// SIMATIC S7-200 SMART project (STEP 7-Micro/WIN SMART), CPU SR30

ORGANIZATION_BLOCK 主程序:OB1
TITLE=程序注释
BEGIN
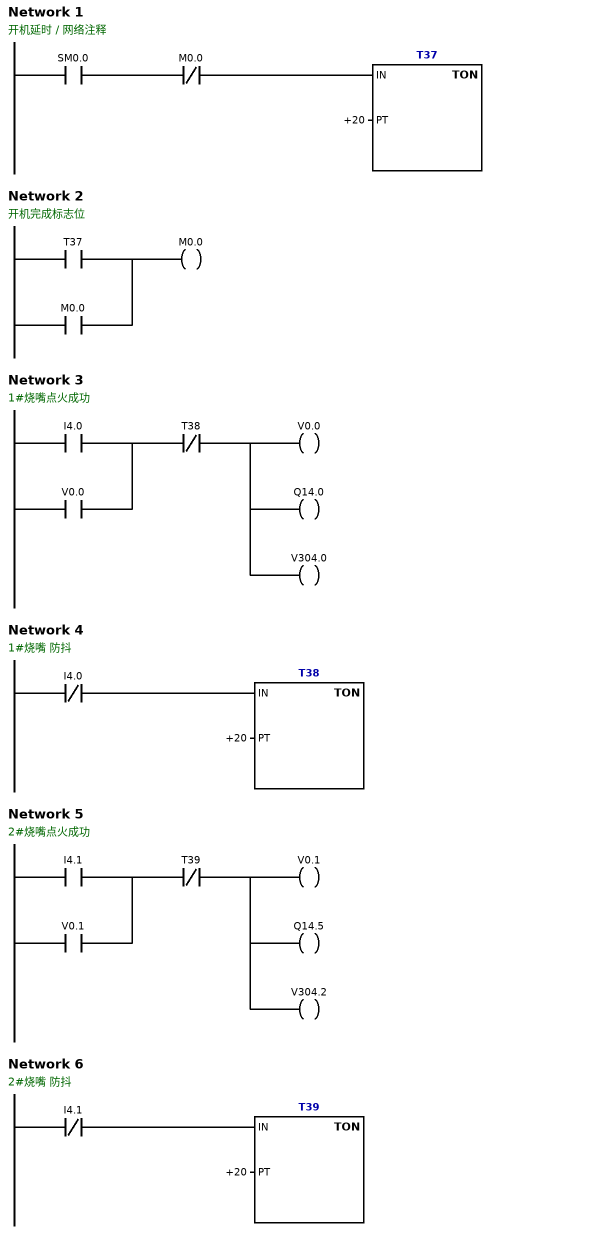
Network 1
// 开机延时
// 网络注释
LD     SM0.0
AN     M0.0
TON    T37, +20
Network 2
// 开机完成标志位
LD     T37
O      M0.0
=      M0.0
Network 3
// 1#烧嘴点火成功
LD     I4.0
O      V0.0
AN     T38
=      V0.0
=      Q14.0
=      V304.0
Network 4
// 1#烧嘴 防抖
LDN    I4.0
TON    T38, +20
Network 5
// 2#烧嘴点火成功
LD     I4.1
O      V0.1
AN     T39
=      V0.1
=      Q14.5
=      V304.2
Network 6
// 2#烧嘴 防抖
LDN    I4.1
TON    T39, +20
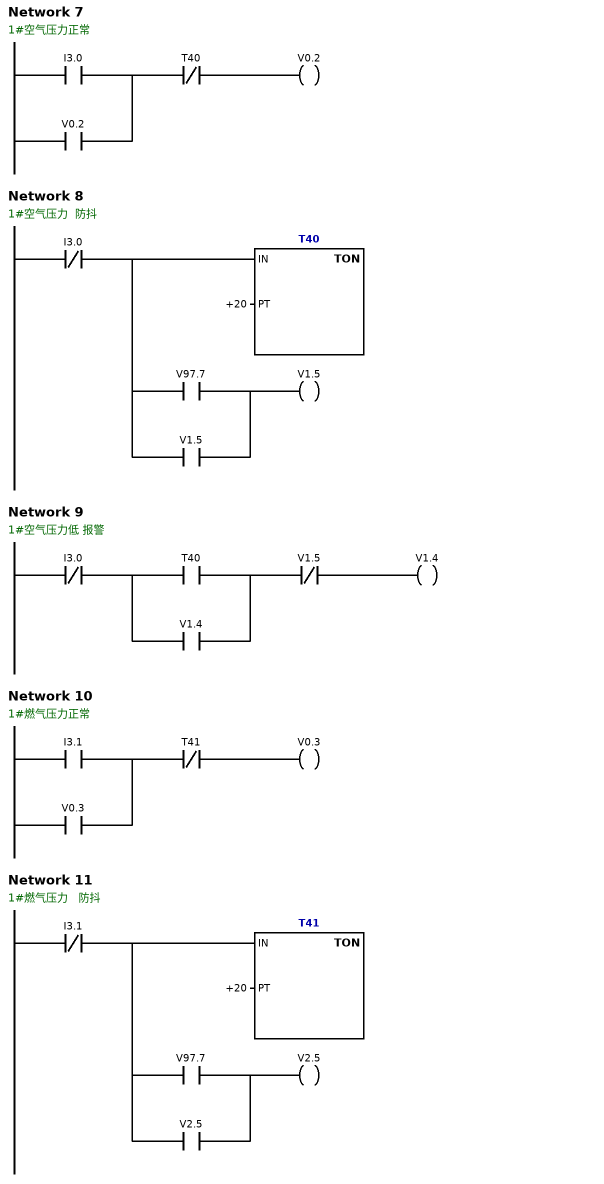
Network 7
// 1#空气压力正常
LD     I3.0
O      V0.2
AN     T40
=      V0.2
Network 8
// 1#空气压力  防抖
LDN    I3.0
TON    T40, +20
LD     V97.7
O      V1.5
ALD
=      V1.5
Network 9
// 1#空气压力低 报警
LDN    I3.0
LD     T40
O      V1.4
ALD
AN     V1.5
=      V1.4
Network 10
// 1#燃气压力正常
LD     I3.1
O      V0.3
AN     T41
=      V0.3
Network 11
// 1#燃气压力   防抖
LDN    I3.1
TON    T41, +20
LD     V97.7
O      V2.5
ALD
=      V2.5
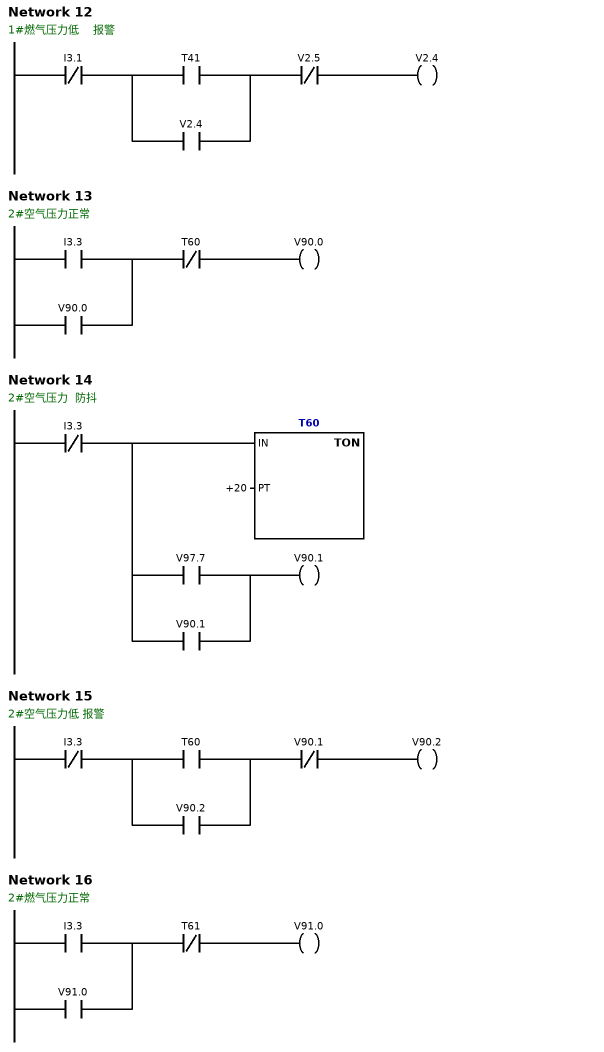
Network 12
// 1#燃气压力低    报警
LDN    I3.1
LD     T41
O      V2.4
ALD
AN     V2.5
=      V2.4
Network 13
// 2#空气压力正常
LD     I3.3
O      V90.0
AN     T60
=      V90.0
Network 14
// 2#空气压力  防抖
LDN    I3.3
TON    T60, +20
LD     V97.7
O      V90.1
ALD
=      V90.1
Network 15
// 2#空气压力低 报警
LDN    I3.3
LD     T60
O      V90.2
ALD
AN     V90.1
=      V90.2
Network 16
// 2#燃气压力正常
LD     I3.3
O      V91.0
AN     T61
=      V91.0
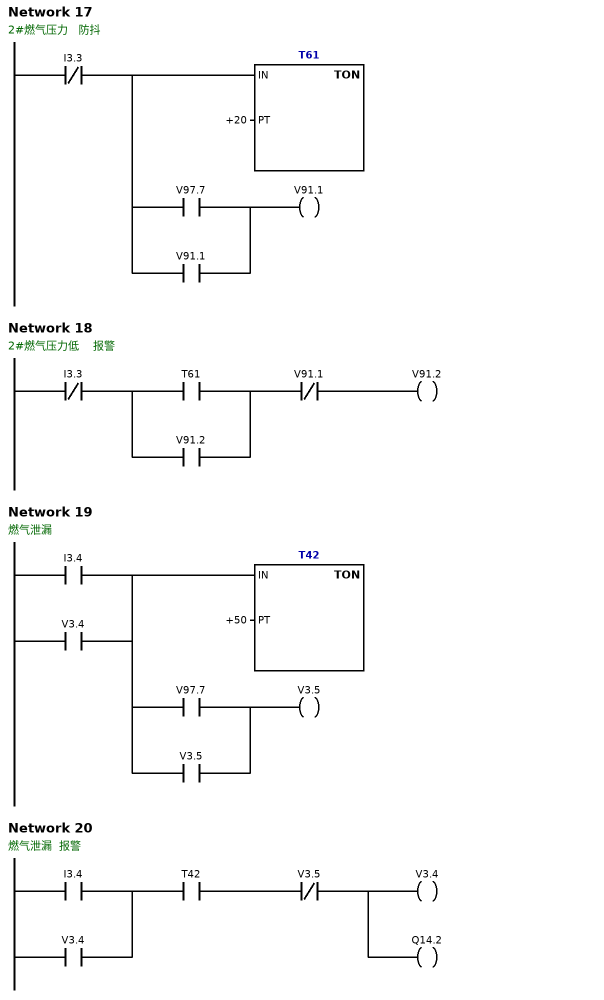
Network 17
// 2#燃气压力   防抖
LDN    I3.3
TON    T61, +20
LD     V97.7
O      V91.1
ALD
=      V91.1
Network 18
// 2#燃气压力低    报警
LDN    I3.3
LD     T61
O      V91.2
ALD
AN     V91.1
=      V91.2
Network 19
// 燃气泄漏
LD     I3.4
O      V3.4
TON    T42, +50
LD     V97.7
O      V3.5
ALD
=      V3.5
Network 20
// 燃气泄漏  报警
LD     I3.4
O      V3.4
A      T42
AN     V3.5
=      V3.4
=      Q14.2
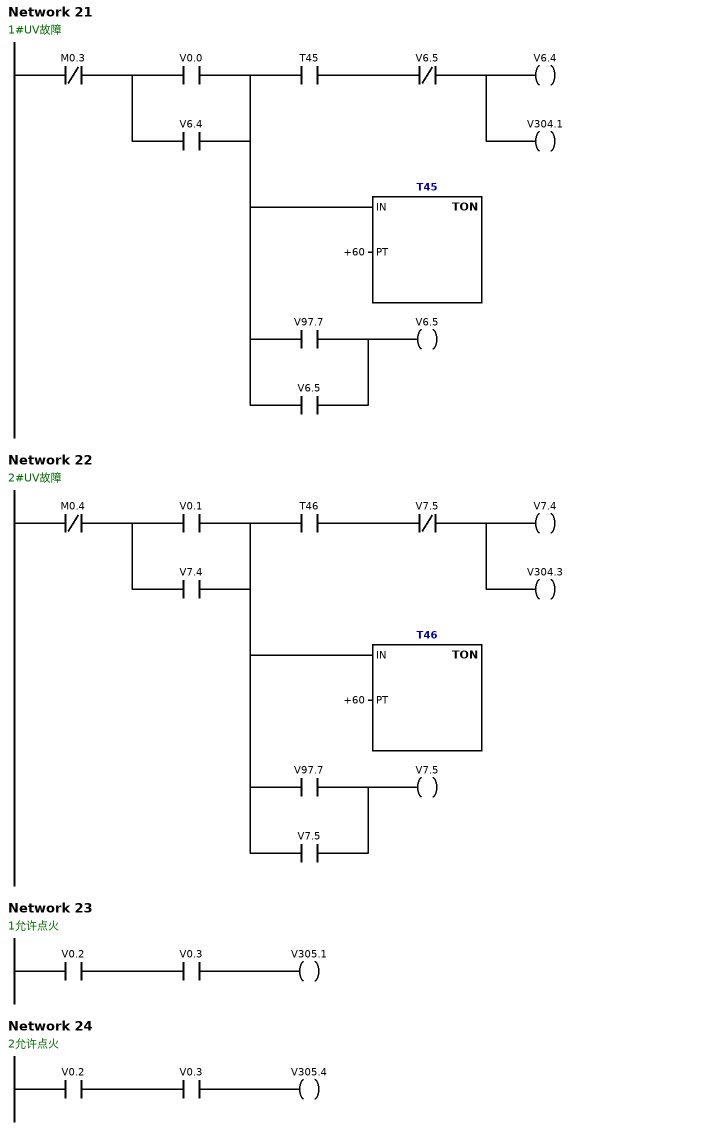
Network 21
// 1#UV故障
LDN    M0.3
LD     V0.0
O      V6.4
ALD
LPS
A      T45
AN     V6.5
=      V6.4
=      V304.1
LRD
TON    T45, +60
LPP
LD     V97.7
O      V6.5
ALD
=      V6.5
Network 22
// 2#UV故障
LDN    M0.4
LD     V0.1
O      V7.4
ALD
LPS
A      T46
AN     V7.5
=      V7.4
=      V304.3
LRD
TON    T46, +60
LPP
LD     V97.7
O      V7.5
ALD
=      V7.5
Network 23
// 1允许点火
// (network saved uncompiled; LAD cells follow)
// row 0: c0 -| |- V0.2  c1 -| |- V0.3  c2 -( ) V305.1
Network 24
// 2允许点火
// (network saved uncompiled; LAD cells follow)
// row 0: c0 -| |- V0.2  c1 -| |- V0.3  c2 -( ) V305.4
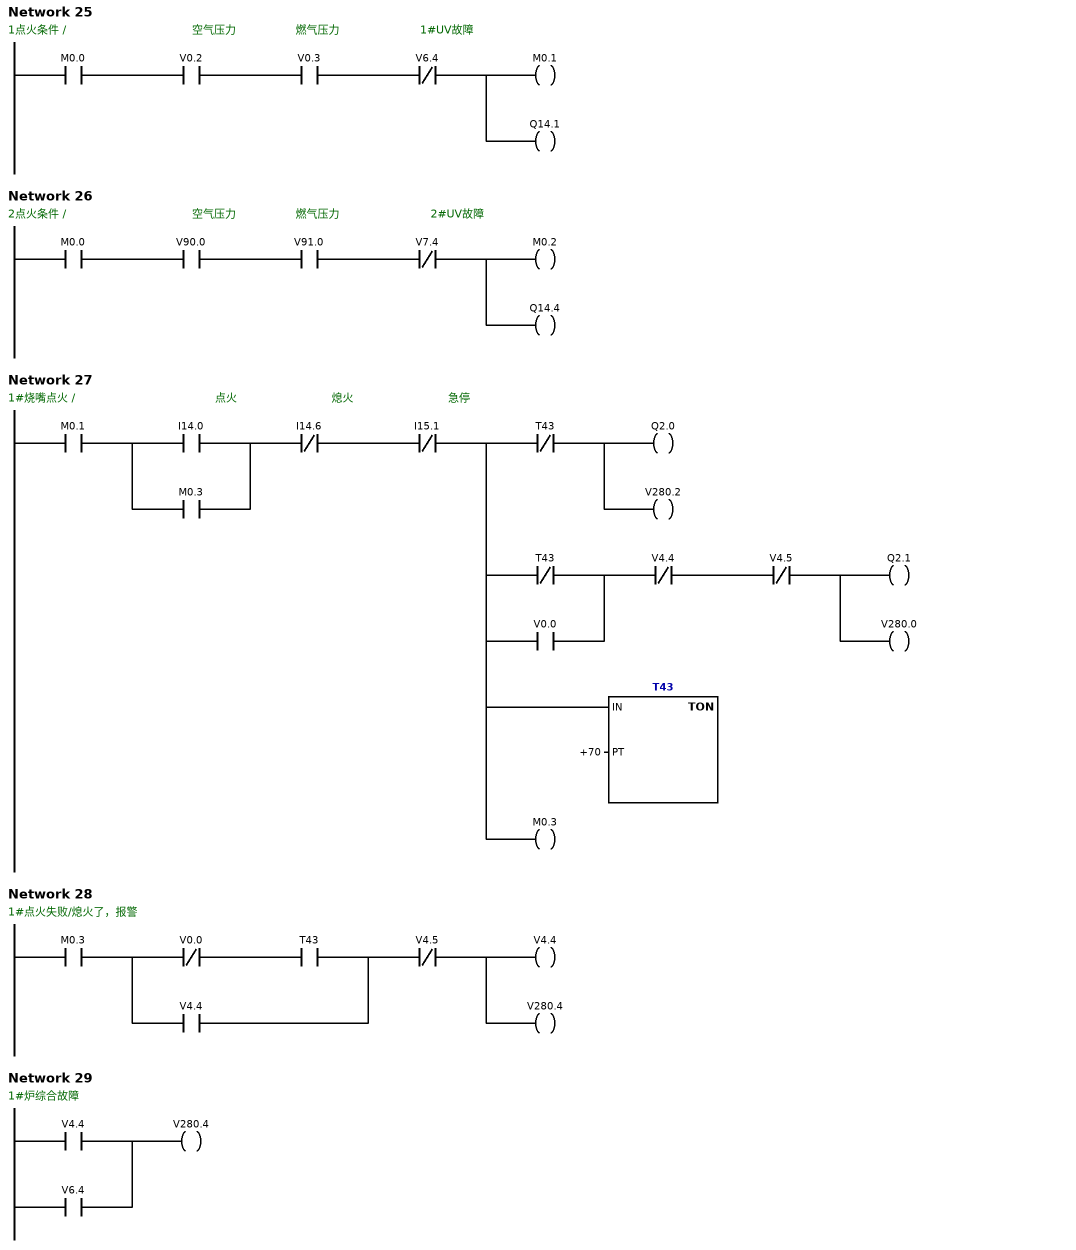
Network 25
// 1点火条件
//                                    空气压力                 燃气压力                       1#UV故障
LD     M0.0
A      V0.2
A      V0.3
AN     V6.4
=      M0.1
=      Q14.1
Network 26
// 2点火条件
//                                    空气压力                 燃气压力                          2#UV故障
LD     M0.0
A      V90.0
A      V91.0
AN     V7.4
=      M0.2
=      Q14.4
Network 27
// 1#烧嘴点火
//                                        点火                           熄火                           急停
LD     M0.1
LD     I14.0
O      M0.3
ALD
AN     I14.6
AN     I15.1
LPS
AN     T43
=      Q2.0
=      V280.2
LRD
LDN    T43
O      V0.0
AN     V4.4
AN     V4.5
ALD
=      Q2.1
=      V280.0
LPP
TON    T43, +70
=      M0.3
Network 28
// 1#点火失败/熄火了，报警
// (network saved uncompiled; LAD cells follow)
// row 0: c0 -| |- M0.3 v  c1 -|/|- V0.0  c2 -| |- T43 v  c3 -|/|- V4.5 v  c4 -( ) V4.4
// row 1: c0 ^  c1 -| |- V4.4  c2 -- ^  c3 ^  c4 -( ) V280.4
Network 29
// 1#炉综合故障
LD     V4.4
O      V6.4
=      V280.4
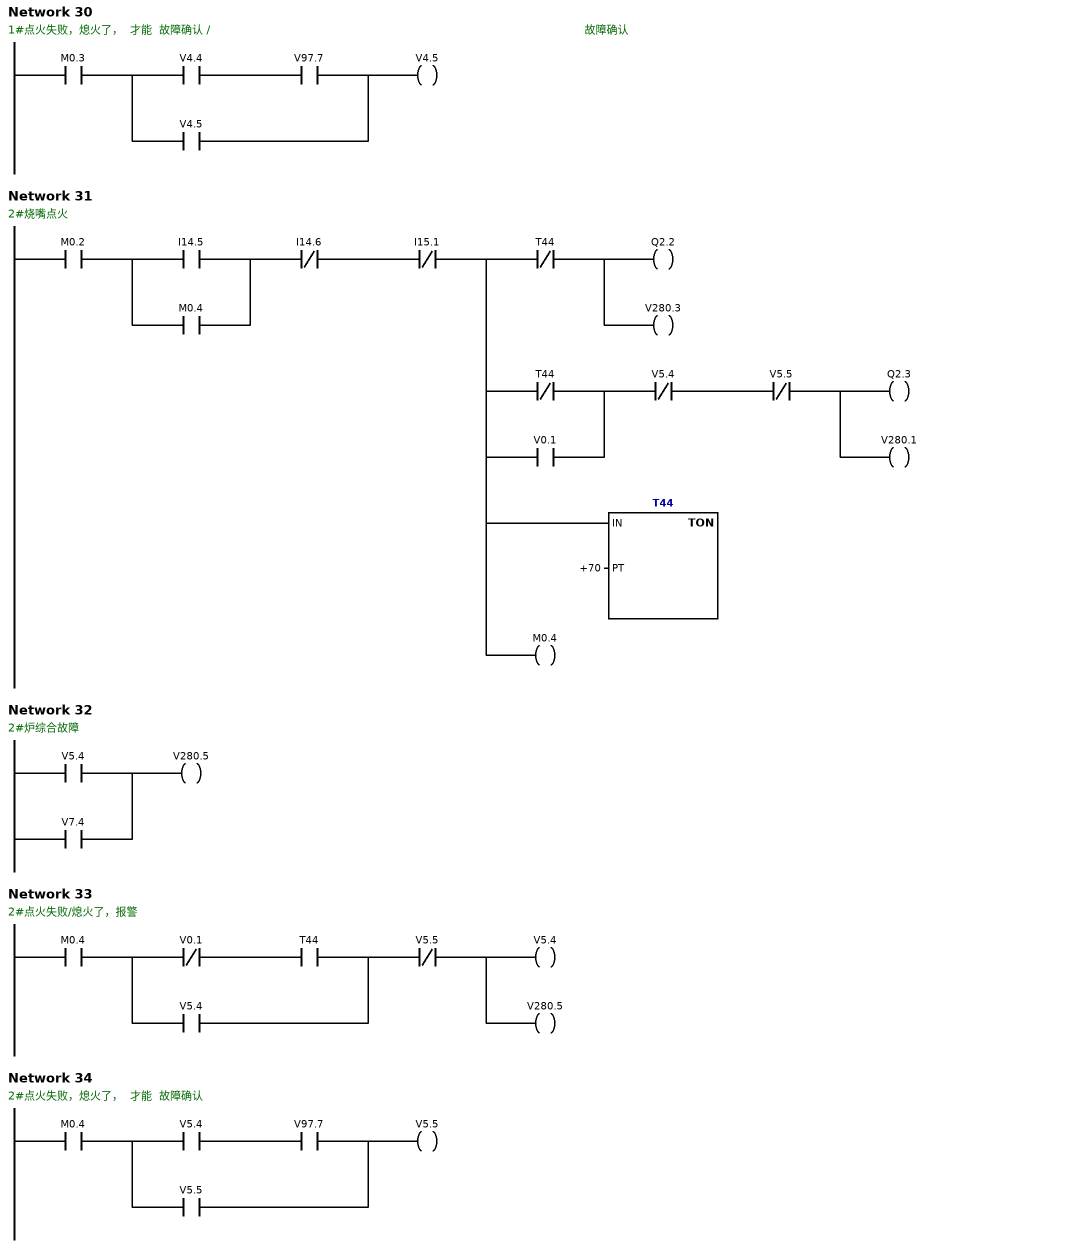
Network 30
// 1#点火失败，熄火了，  才能  故障确认
//                                                                                                           故障确认
LD     M0.3
LD     V4.4
A      V97.7
O      V4.5
ALD
=      V4.5
Network 31
// 2#烧嘴点火
// (network saved uncompiled; LAD cells follow)
// row 0: c0 -| |- M0.2 v  c1 -| |- I14.5 v  c2 -|/|- I14.6  c3 -|/|- I15.1 v  c4 -|/|- T44 v  c5 -( ) Q2.2
// row 1: c0 ^  c1 -| |- M0.4 ^  c3 ^v  c4 ^  c5 -( ) V280.3
// row 2: c3 ^v  c4 -|/|- T44 v  c5 -|/|- V5.4  c6 -|/|- V5.5 v  c7 -( ) Q2.3
// row 3: c3 ^v  c4 -| |- V0.1 ^  c6 ^  c7 -( ) V280.1
// row 4: c3 ^v  c4 --  c5 [TON T44 IN:=power@row4, PT:=+70]
// row 5: c3 ^v  c5 [box]
// row 6: c3 ^  c4 -( ) M0.4
Network 32
// 2#炉综合故障
LD     V5.4
O      V7.4
=      V280.5
Network 33
// 2#点火失败/熄火了，报警
// (network saved uncompiled; LAD cells follow)
// row 0: c0 -| |- M0.4 v  c1 -|/|- V0.1  c2 -| |- T44 v  c3 -|/|- V5.5 v  c4 -( ) V5.4
// row 1: c0 ^  c1 -| |- V5.4  c2 -- ^  c3 ^  c4 -( ) V280.5
Network 34
// 2#点火失败，熄火了，  才能  故障确认
LD     M0.4
LD     V5.4
A      V97.7
O      V5.5
ALD
=      V5.5
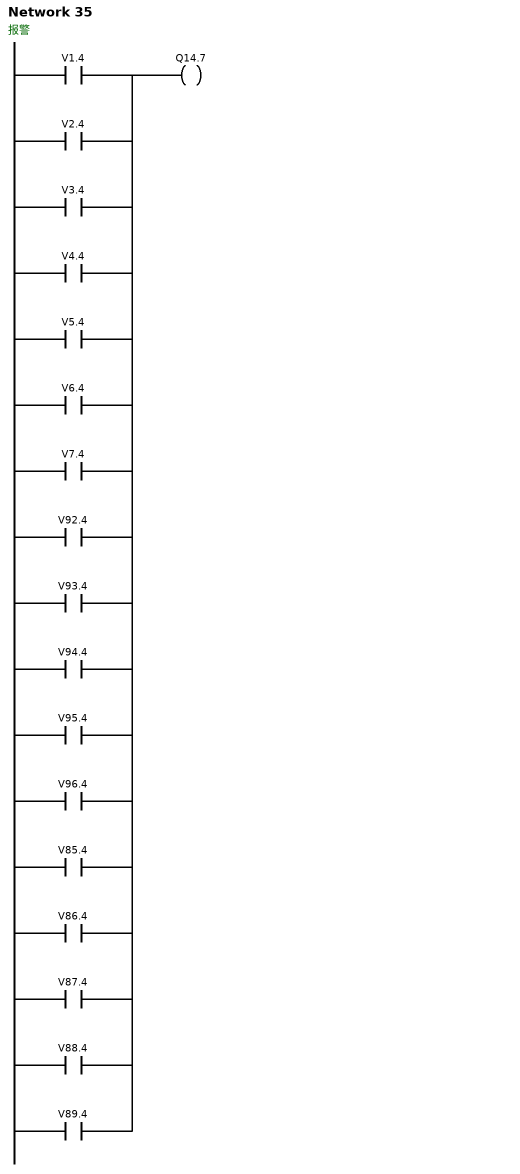
Network 35
// 报警
LD     V1.4
O      V2.4
O      V3.4
O      V4.4
O      V5.4
O      V6.4
O      V7.4
O      V92.4
O      V93.4
O      V94.4
O      V95.4
O      V96.4
O      V85.4
O      V86.4
O      V87.4
O      V88.4
O      V89.4
=      Q14.7
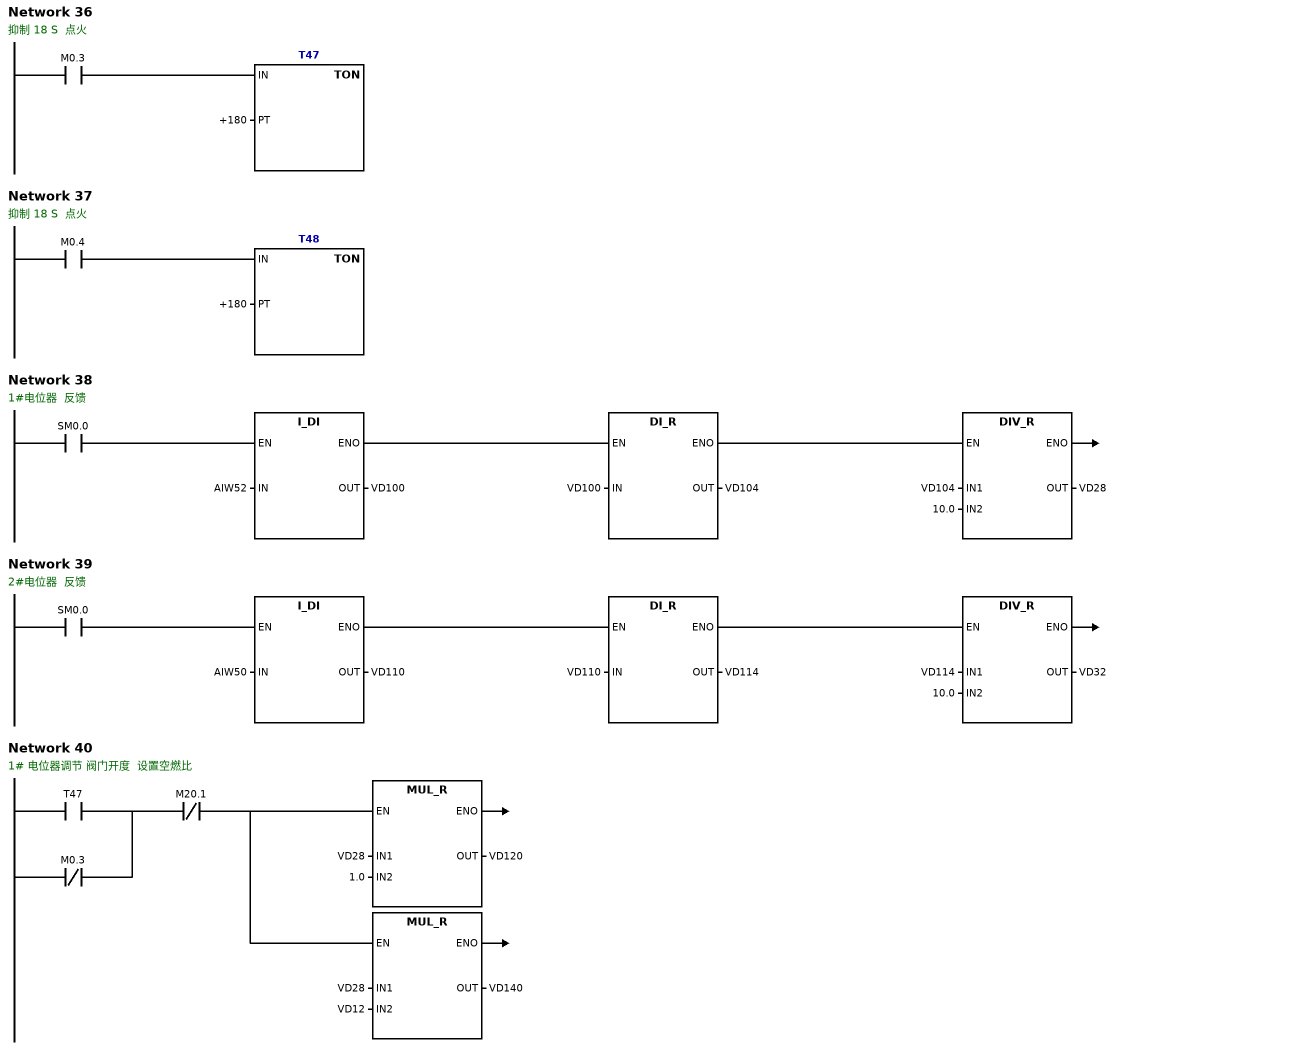
Network 36
// 抑制 18 S  点火
LD     M0.3
TON    T47, +180
Network 37
// 抑制 18 S  点火
LD     M0.4
TON    T48, +180
Network 38
// 1#电位器  反馈
LD     SM0.0
ITD    AIW52, VD100
AENO
DTR    VD100, VD104
AENO
MOVR   VD104, VD28
/R     10.0, VD28
Network 39
// 2#电位器  反馈
LD     SM0.0
ITD    AIW50, VD110
AENO
DTR    VD110, VD114
AENO
MOVR   VD114, VD32
/R     10.0, VD32
Network 40
// 1# 电位器调节 阀门开度  设置空燃比
LD     T47
ON     M0.3
AN     M20.1
MOVR   VD28, VD120
*R     1.0, VD120
MOVR   VD28, VD140
*R     VD12, VD140
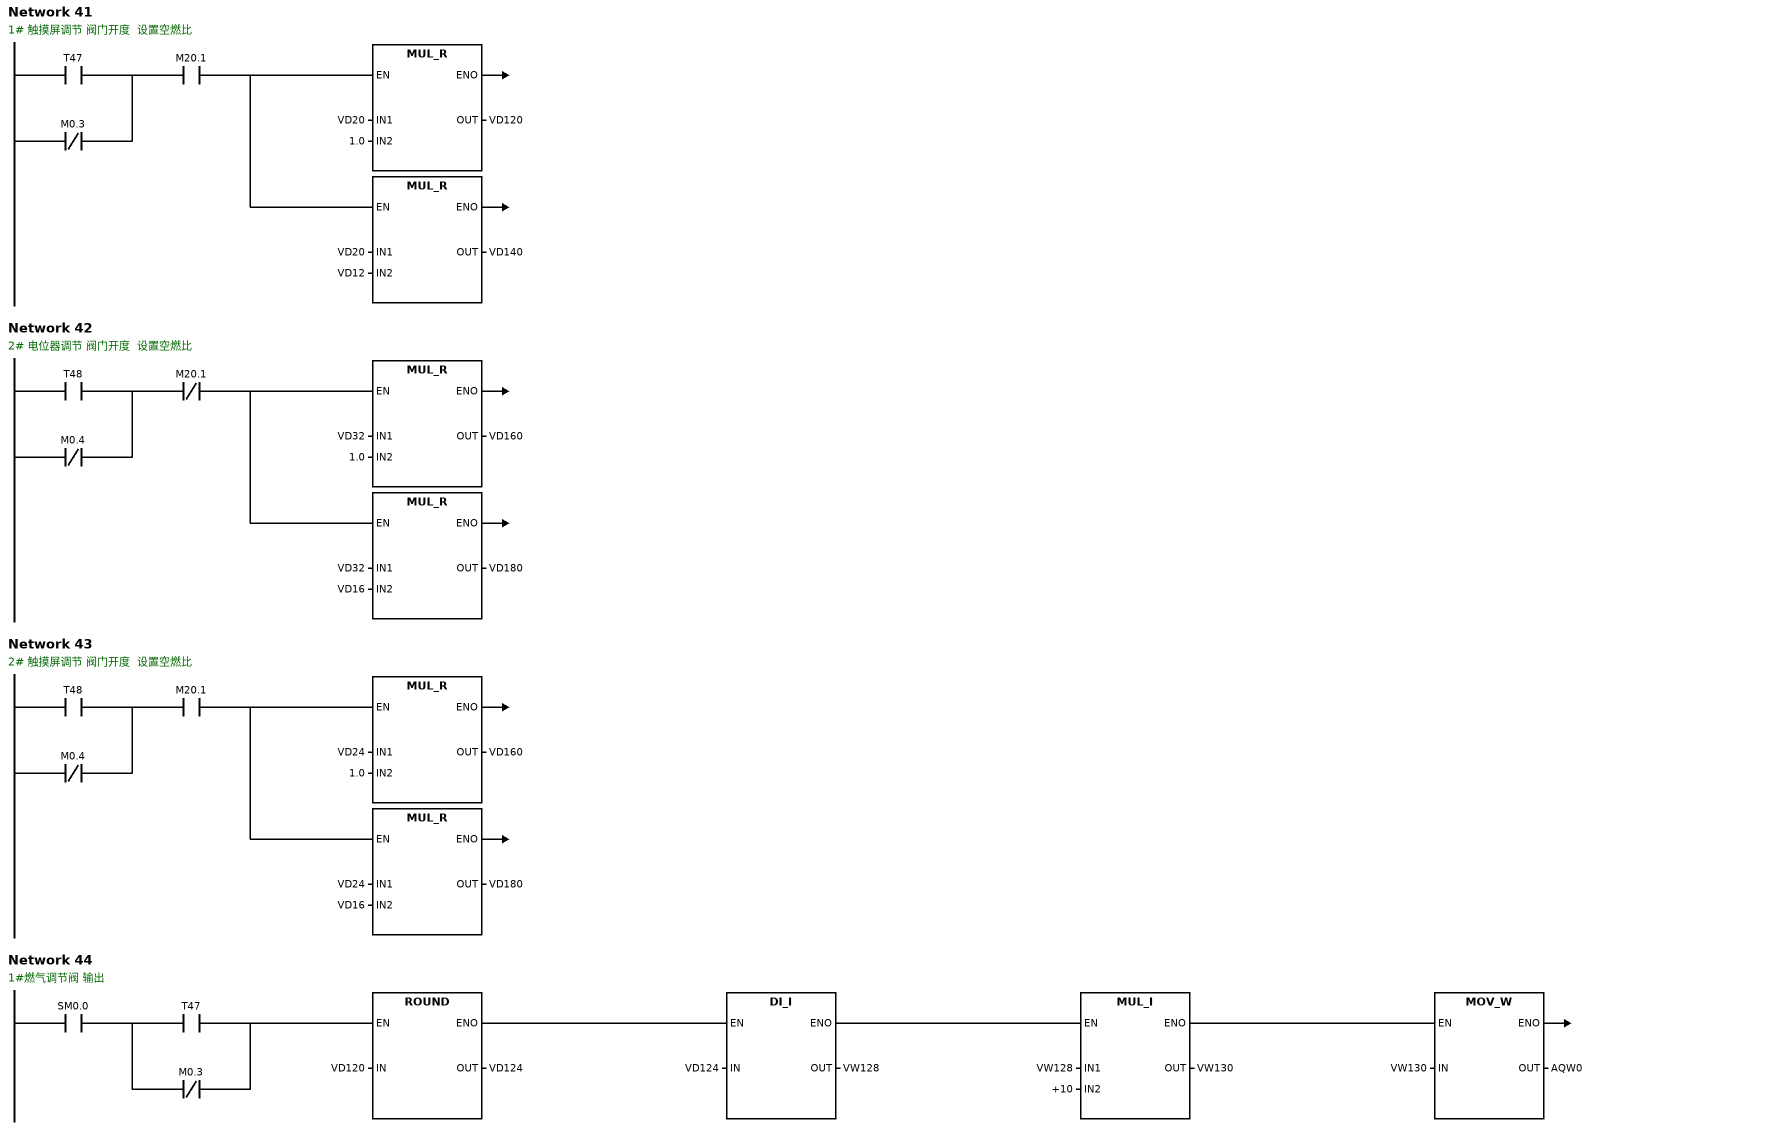
Network 41
// 1# 触摸屏调节 阀门开度  设置空燃比
LD     T47
ON     M0.3
A      M20.1
MOVR   VD20, VD120
*R     1.0, VD120
MOVR   VD20, VD140
*R     VD12, VD140
Network 42
// 2# 电位器调节 阀门开度  设置空燃比
LD     T48
ON     M0.4
AN     M20.1
MOVR   VD32, VD160
*R     1.0, VD160
MOVR   VD32, VD180
*R     VD16, VD180
Network 43
// 2# 触摸屏调节 阀门开度  设置空燃比
LD     T48
ON     M0.4
A      M20.1
MOVR   VD24, VD160
*R     1.0, VD160
MOVR   VD24, VD180
*R     VD16, VD180
Network 44
// 1#燃气调节阀 输出
LD     SM0.0
LD     T47
ON     M0.3
ALD
ROUND  VD120, VD124
AENO
DTI    VD124, VW128
AENO
MOVW   VW128, VW130
AENO
*I     +10, VW130
AENO
MOVW   VW130, AQW0
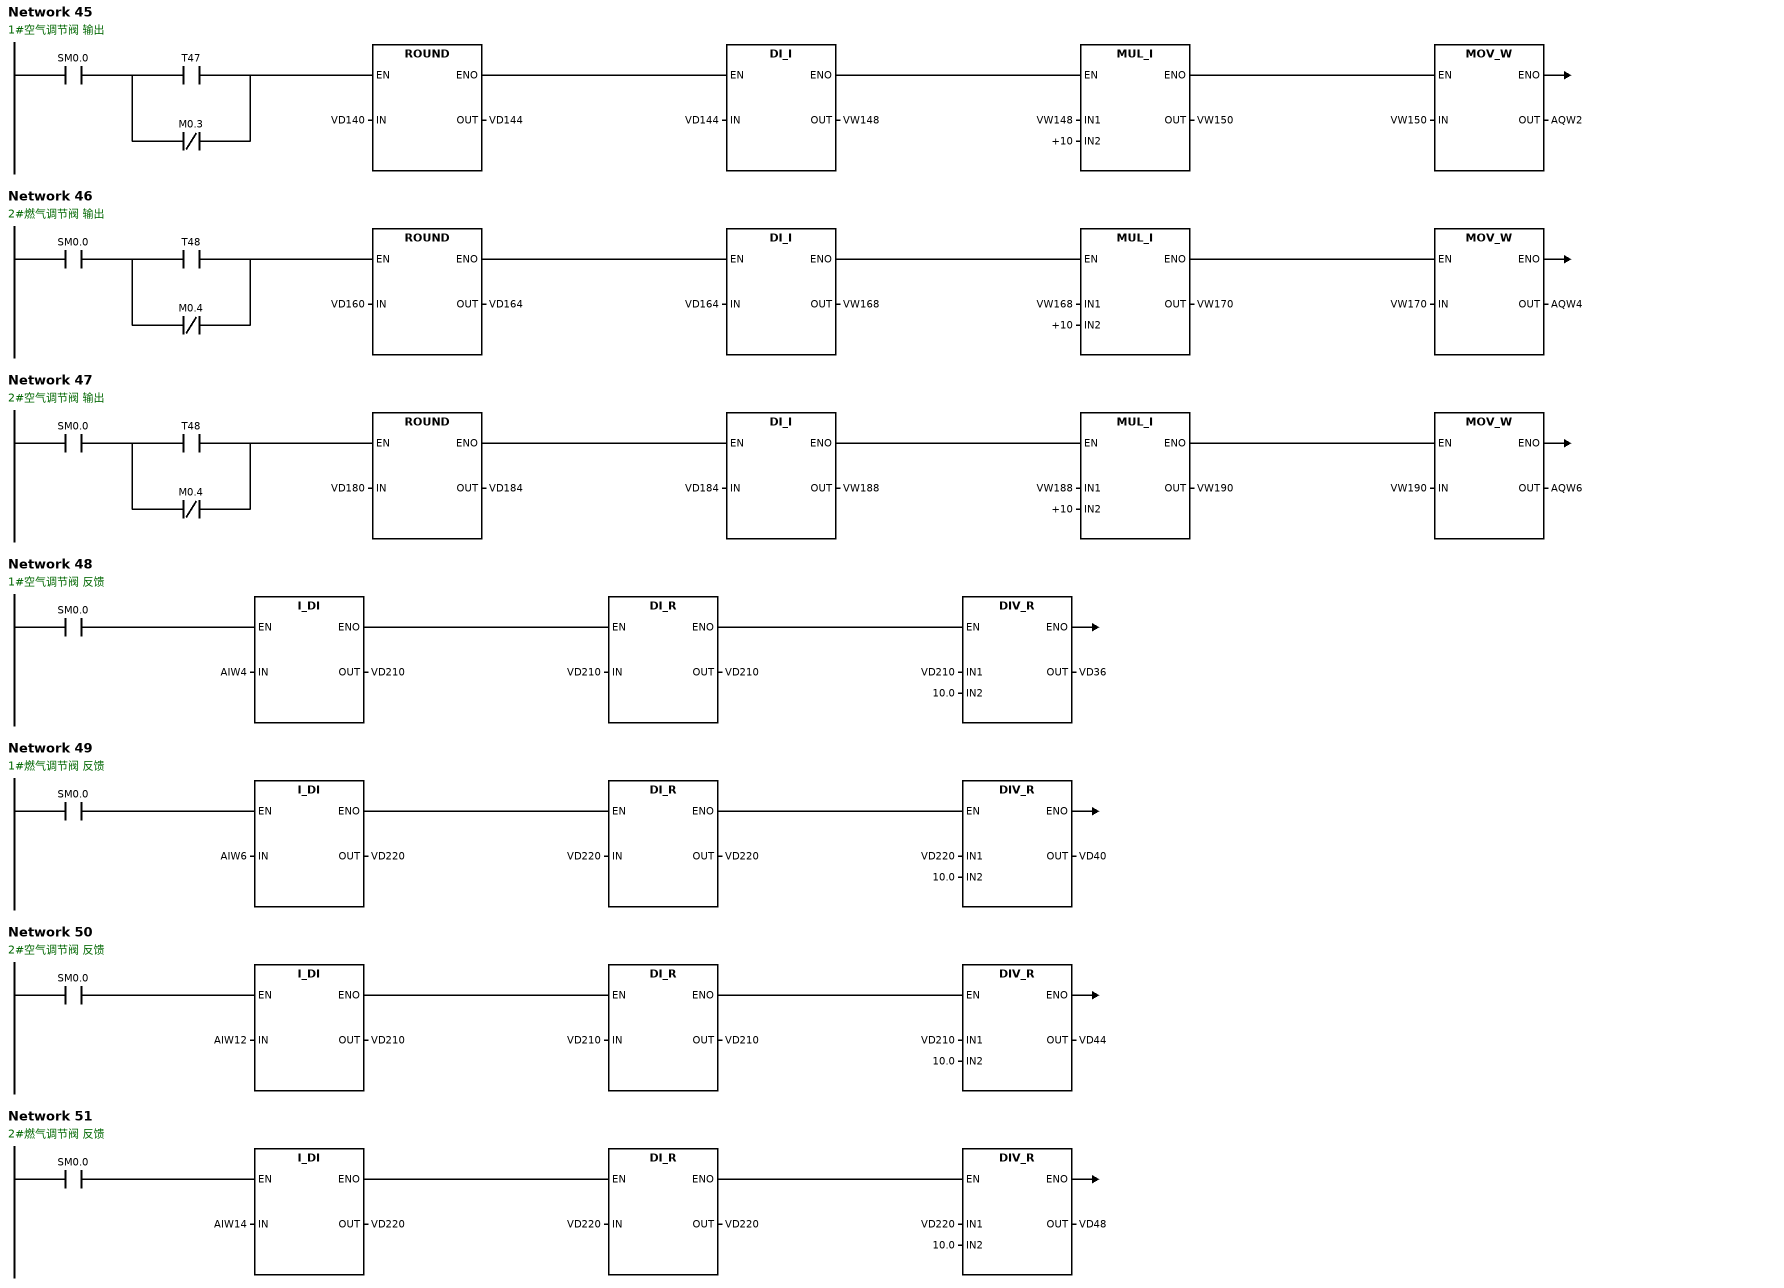
Network 45
// 1#空气调节阀 输出
LD     SM0.0
LD     T47
ON     M0.3
ALD
ROUND  VD140, VD144
AENO
DTI    VD144, VW148
AENO
MOVW   VW148, VW150
AENO
*I     +10, VW150
AENO
MOVW   VW150, AQW2
Network 46
// 2#燃气调节阀 输出
LD     SM0.0
LD     T48
ON     M0.4
ALD
ROUND  VD160, VD164
AENO
DTI    VD164, VW168
AENO
MOVW   VW168, VW170
AENO
*I     +10, VW170
AENO
MOVW   VW170, AQW4
Network 47
// 2#空气调节阀 输出
LD     SM0.0
LD     T48
ON     M0.4
ALD
ROUND  VD180, VD184
AENO
DTI    VD184, VW188
AENO
MOVW   VW188, VW190
AENO
*I     +10, VW190
AENO
MOVW   VW190, AQW6
Network 48
// 1#空气调节阀 反馈
LD     SM0.0
ITD    AIW4, VD210
AENO
DTR    VD210, VD210
AENO
MOVR   VD210, VD36
/R     10.0, VD36
Network 49
// 1#燃气调节阀 反馈
LD     SM0.0
ITD    AIW6, VD220
AENO
DTR    VD220, VD220
AENO
MOVR   VD220, VD40
/R     10.0, VD40
Network 50
// 2#空气调节阀 反馈
LD     SM0.0
ITD    AIW12, VD210
AENO
DTR    VD210, VD210
AENO
MOVR   VD210, VD44
/R     10.0, VD44
Network 51
// 2#燃气调节阀 反馈
LD     SM0.0
ITD    AIW14, VD220
AENO
DTR    VD220, VD220
AENO
MOVR   VD220, VD48
/R     10.0, VD48
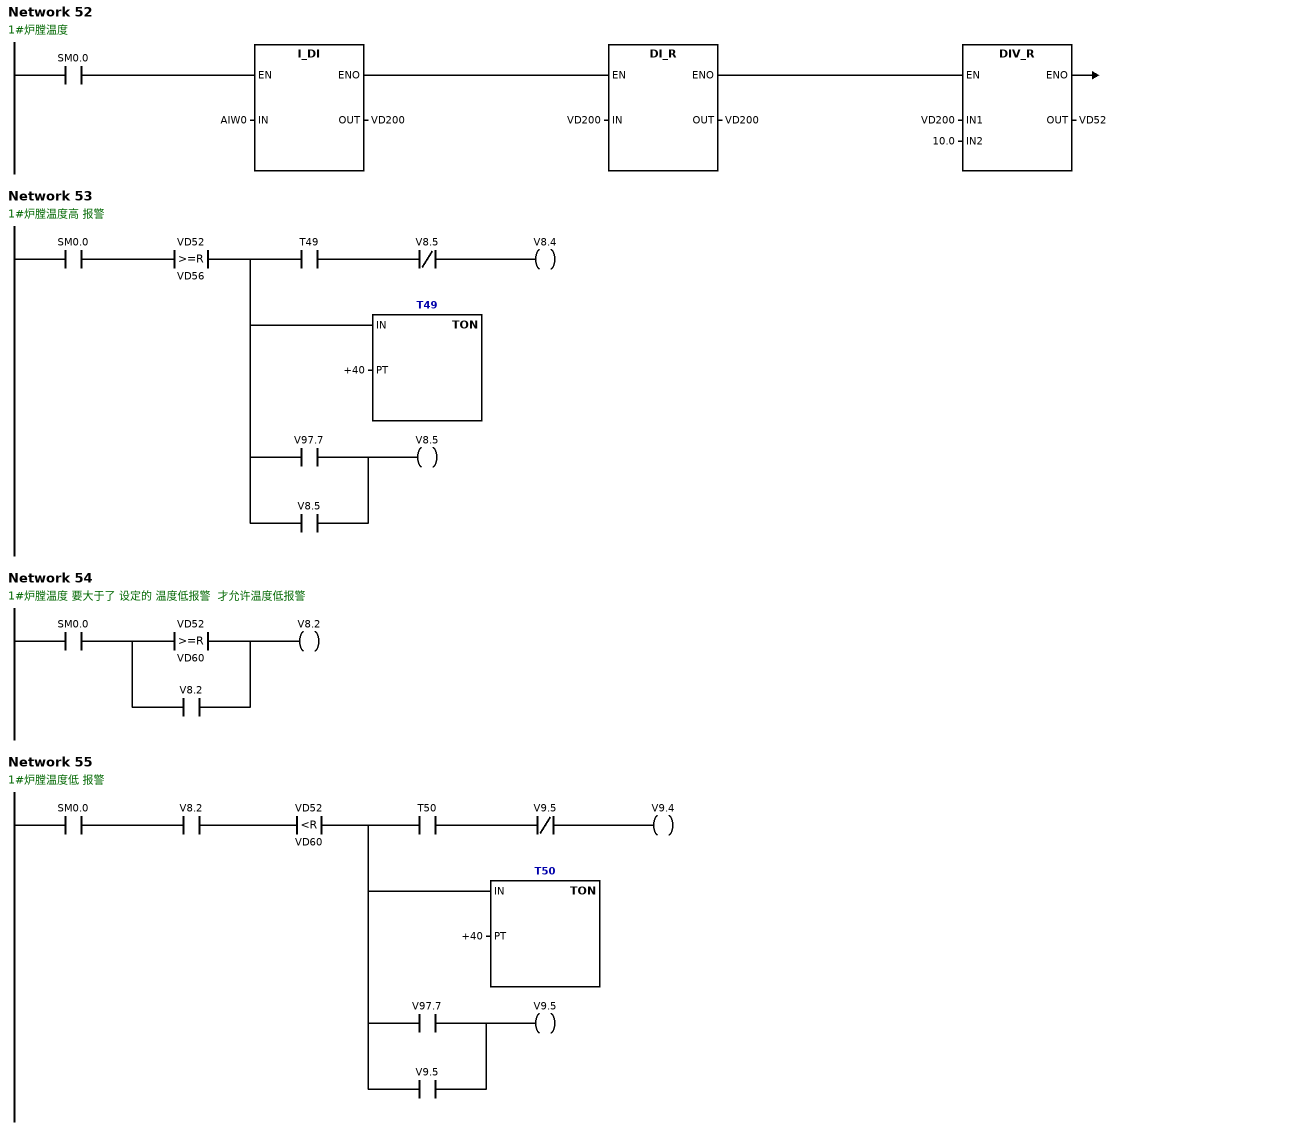
Network 52
// 1#炉膛温度
LD     SM0.0
ITD    AIW0, VD200
AENO
DTR    VD200, VD200
AENO
MOVR   VD200, VD52
/R     10.0, VD52
Network 53
// 1#炉膛温度高 报警
LD     SM0.0
AR>=   VD52, VD56
LPS
A      T49
AN     V8.5
=      V8.4
LRD
TON    T49, +40
LPP
LD     V97.7
O      V8.5
ALD
=      V8.5
Network 54
// 1#炉膛温度 要大于了 设定的 温度低报警  才允许温度低报警
LD     SM0.0
LDR>=  VD52, VD60
O      V8.2
ALD
=      V8.2
Network 55
// 1#炉膛温度低 报警
LD     SM0.0
A      V8.2
AR<    VD52, VD60
LPS
A      T50
AN     V9.5
=      V9.4
LRD
TON    T50, +40
LPP
LD     V97.7
O      V9.5
ALD
=      V9.5
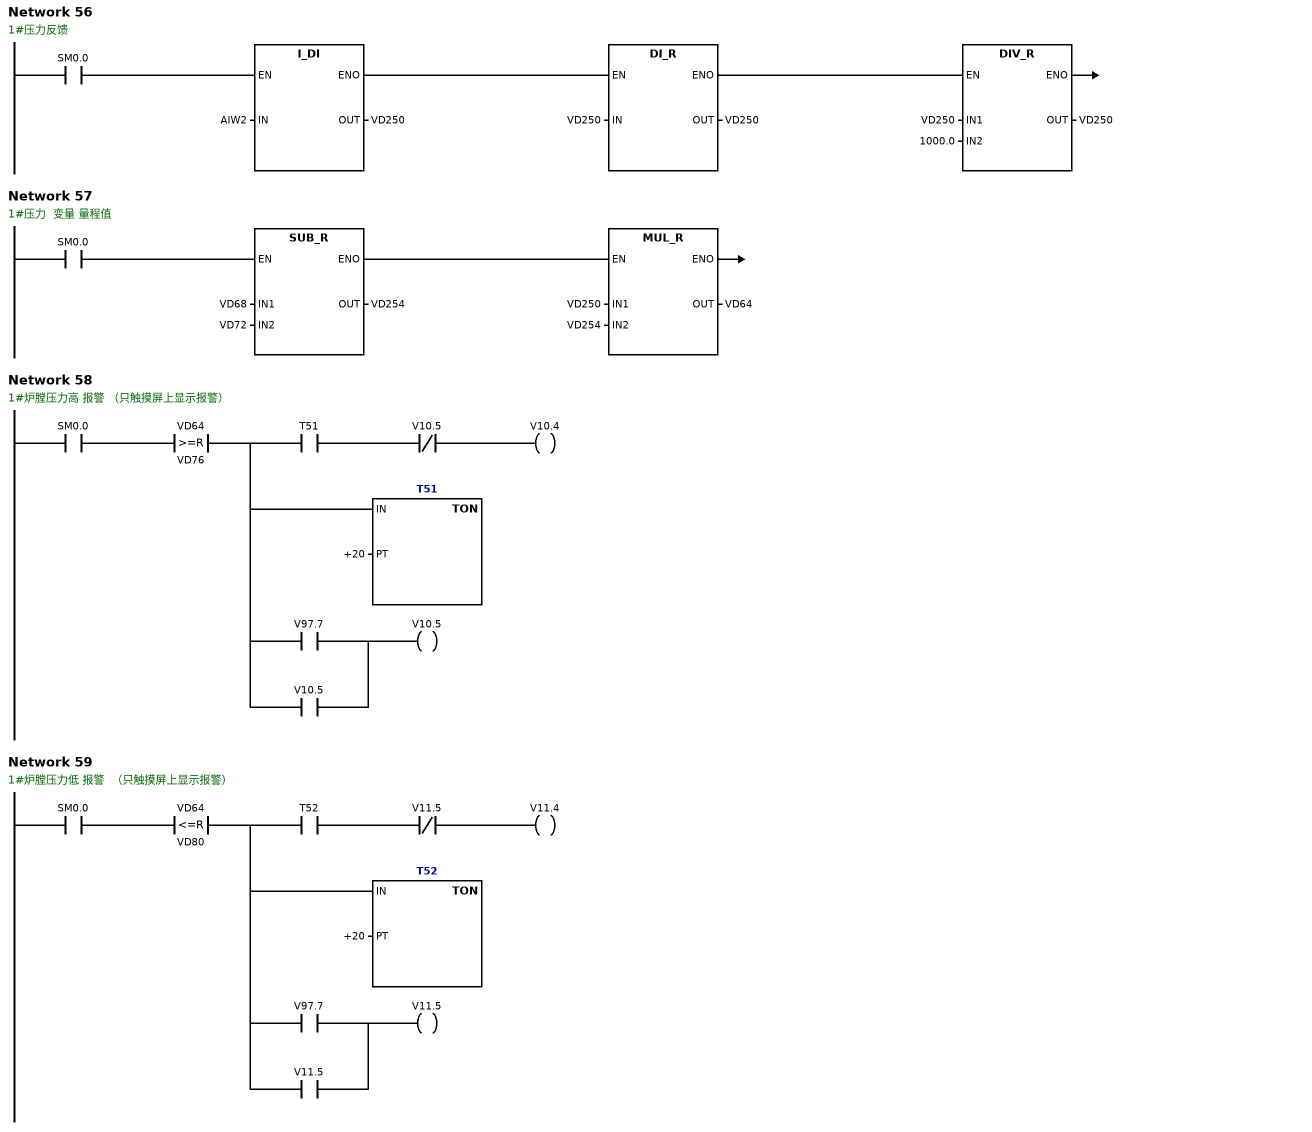
Network 56
// 1#压力反馈
LD     SM0.0
ITD    AIW2, VD250
AENO
DTR    VD250, VD250
AENO
/R     1000.0, VD250
Network 57
// 1#压力  变量 量程值  
LD     SM0.0
MOVR   VD68, VD254
AENO
-R     VD72, VD254
AENO
MOVR   VD250, VD64
*R     VD254, VD64
Network 58
// 1#炉膛压力高 报警 （只触摸屏上显示报警）
LD     SM0.0
AR>=   VD64, VD76
LPS
A      T51
AN     V10.5
=      V10.4
LRD
TON    T51, +20
LPP
LD     V97.7
O      V10.5
ALD
=      V10.5
Network 59
// 1#炉膛压力低 报警  （只触摸屏上显示报警）
LD     SM0.0
AR<=   VD64, VD80
LPS
A      T52
AN     V11.5
=      V11.4
LRD
TON    T52, +20
LPP
LD     V97.7
O      V11.5
ALD
=      V11.5
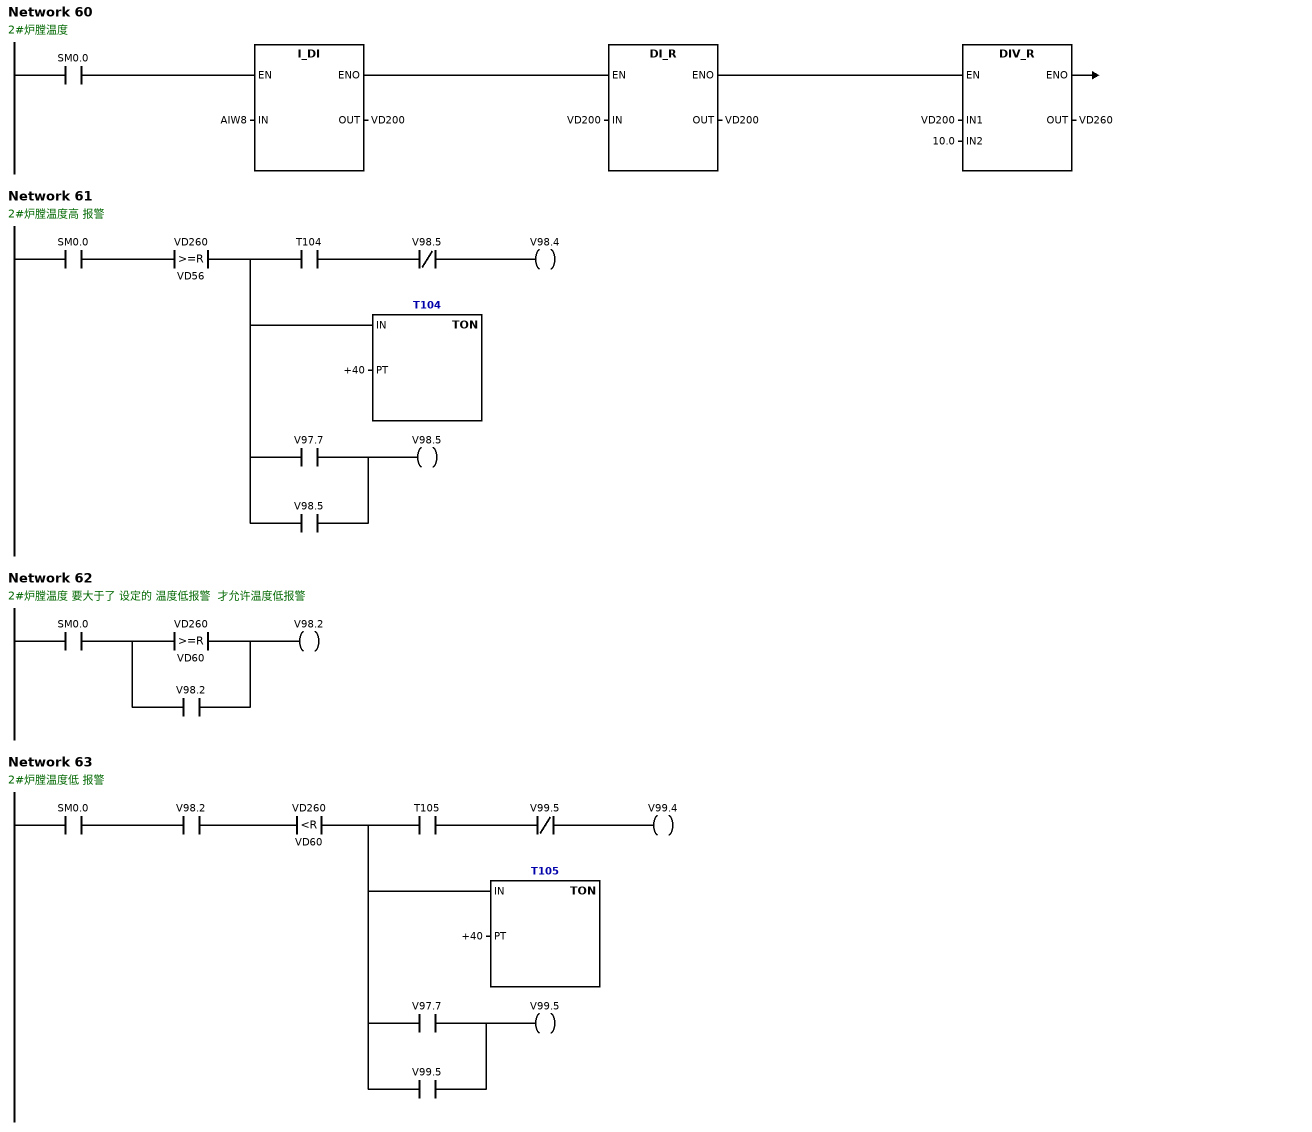
Network 60
// 2#炉膛温度
LD     SM0.0
ITD    AIW8, VD200
AENO
DTR    VD200, VD200
AENO
MOVR   VD200, VD260
/R     10.0, VD260
Network 61
// 2#炉膛温度高 报警
LD     SM0.0
AR>=   VD260, VD56
LPS
A      T104
AN     V98.5
=      V98.4
LRD
TON    T104, +40
LPP
LD     V97.7
O      V98.5
ALD
=      V98.5
Network 62
// 2#炉膛温度 要大于了 设定的 温度低报警  才允许温度低报警
LD     SM0.0
LDR>=  VD260, VD60
O      V98.2
ALD
=      V98.2
Network 63
// 2#炉膛温度低 报警
LD     SM0.0
A      V98.2
AR<    VD260, VD60
LPS
A      T105
AN     V99.5
=      V99.4
LRD
TON    T105, +40
LPP
LD     V97.7
O      V99.5
ALD
=      V99.5
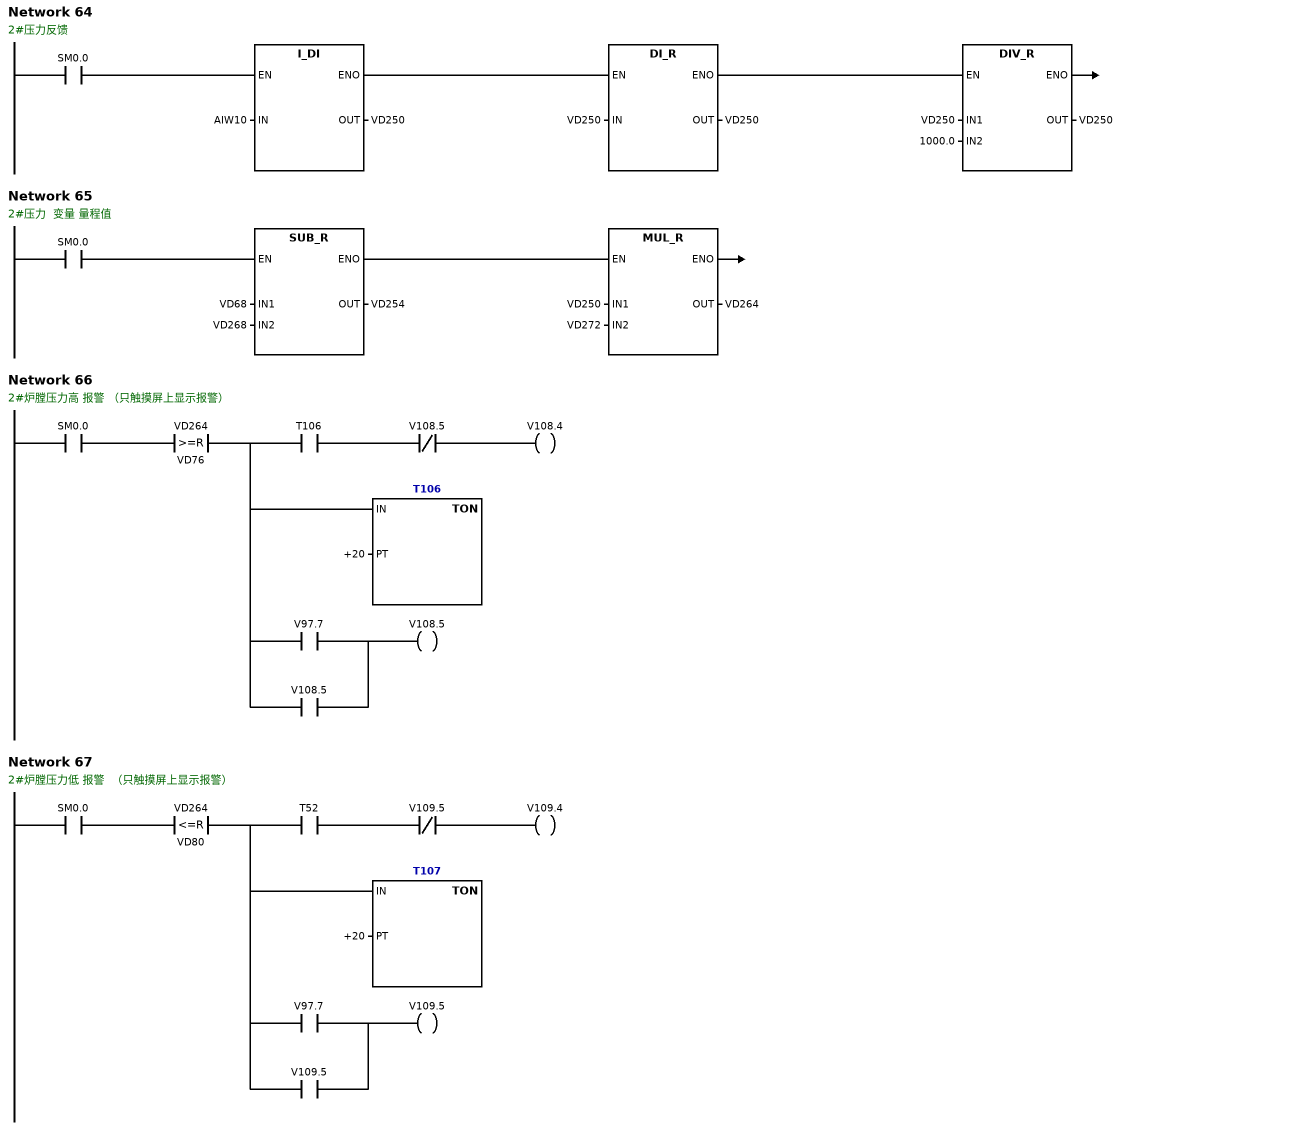
Network 64
// 2#压力反馈
LD     SM0.0
ITD    AIW10, VD250
AENO
DTR    VD250, VD250
AENO
/R     1000.0, VD250
Network 65
// 2#压力  变量 量程值  
LD     SM0.0
MOVR   VD68, VD254
AENO
-R     VD268, VD254
AENO
MOVR   VD250, VD264
*R     VD272, VD264
Network 66
// 2#炉膛压力高 报警 （只触摸屏上显示报警）
LD     SM0.0
AR>=   VD264, VD76
LPS
A      T106
AN     V108.5
=      V108.4
LRD
TON    T106, +20
LPP
LD     V97.7
O      V108.5
ALD
=      V108.5
Network 67
// 2#炉膛压力低 报警  （只触摸屏上显示报警）
LD     SM0.0
AR<=   VD264, VD80
LPS
A      T52
AN     V109.5
=      V109.4
LRD
TON    T107, +20
LPP
LD     V97.7
O      V109.5
ALD
=      V109.5
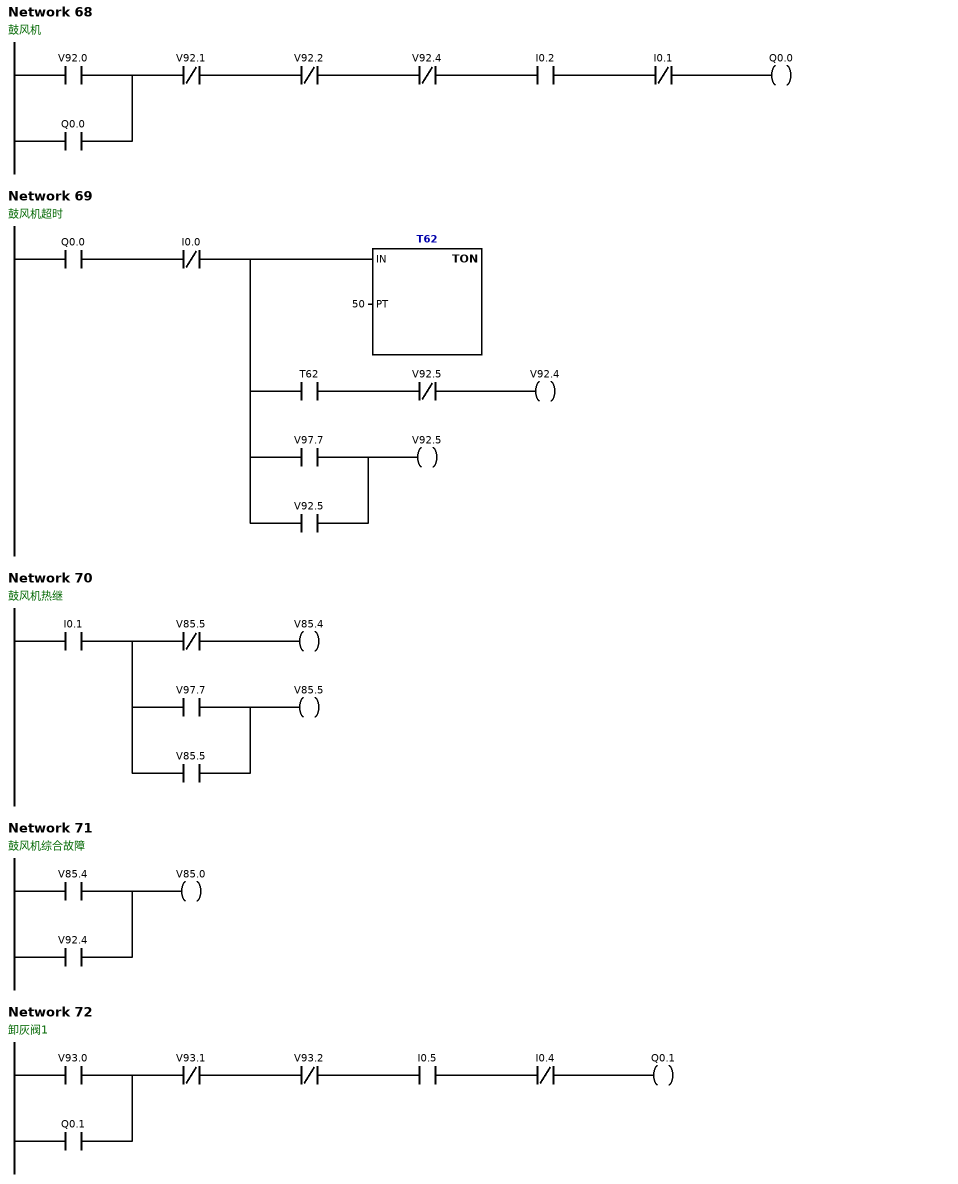
Network 68
// 鼓风机
// (network saved uncompiled; LAD cells follow)
// row 0: c0 -| |- V92.0 v  c1 -|/|- V92.1  c2 -|/|- V92.2  c3 -|/|- V92.4  c4 -| |- I0.2  c5 -|/|- I0.1  c6 -( ) Q0.0
// row 1: c0 -| |- Q0.0 ^
Network 69
// 鼓风机超时
// (network saved uncompiled; LAD cells follow)
// row 0: c0 -| |- Q0.0  c1 -|/|- I0.0 v  c2 --  c3 [TON T62 IN:=power@row0, PT:=50]
// row 1: c1 ^v  c3 [box]
// row 2: c1 ^v  c2 -| |- T62  c3 -|/|- V92.5  c4 -( ) V92.4
// row 3: c1 ^v  c2 -| |- V97.7 v  c3 -( ) V92.5
// row 4: c1 ^  c2 -| |- V92.5 ^
Network 70
// 鼓风机热继
LD     I0.1
LPS
AN     V85.5
=      V85.4
LPP
LD     V97.7
O      V85.5
ALD
=      V85.5
Network 71
// 鼓风机综合故障
// (network saved uncompiled; LAD cells follow)
// row 0: c0 -| |- V85.4 v  c1 -( ) V85.0
// row 1: c0 -| |- V92.4 ^
Network 72
// 卸灰阀1
LD     V93.0
O      Q0.1
AN     V93.1
AN     V93.2
A      I0.5
AN     I0.4
=      Q0.1
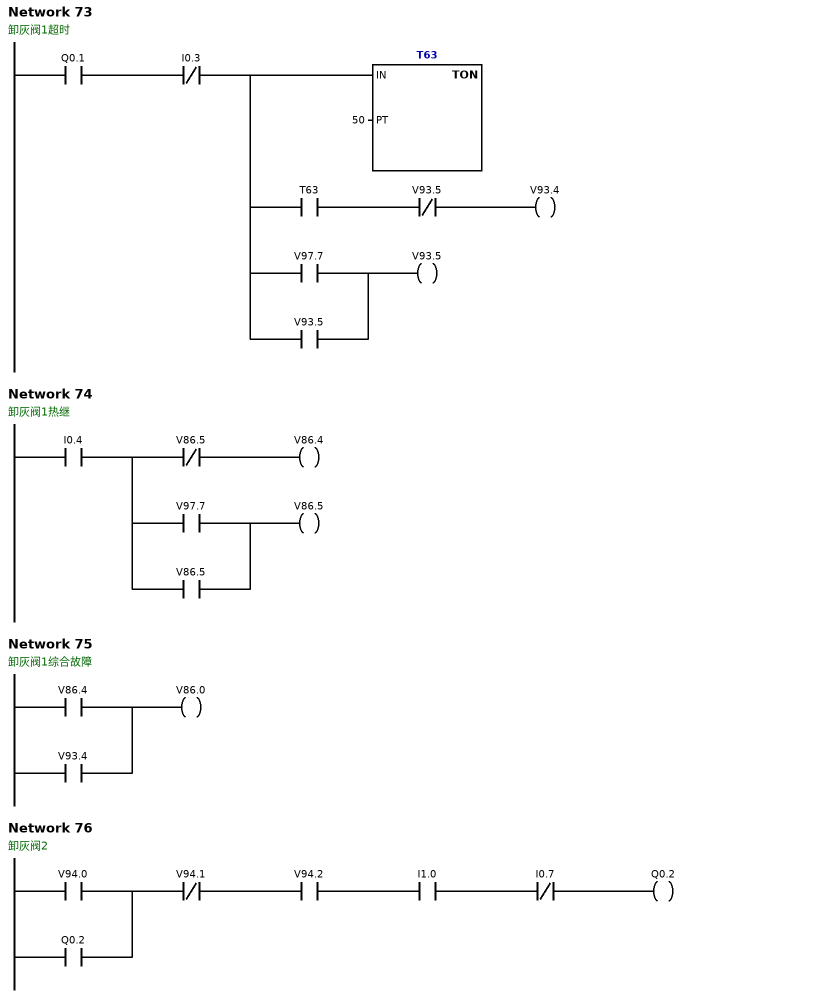
Network 73
// 卸灰阀1超时
LD     Q0.1
AN     I0.3
LPS
TON    T63, 50
A      T63
AN     V93.5
=      V93.4
LPP
LD     V97.7
O      V93.5
ALD
=      V93.5
Network 74
// 卸灰阀1热继
LD     I0.4
LPS
AN     V86.5
=      V86.4
LPP
LD     V97.7
O      V86.5
ALD
=      V86.5
Network 75
// 卸灰阀1综合故障
LD     V86.4
O      V93.4
=      V86.0
Network 76
// 卸灰阀2
LD     V94.0
O      Q0.2
AN     V94.1
A      V94.2
A      I1.0
AN     I0.7
=      Q0.2
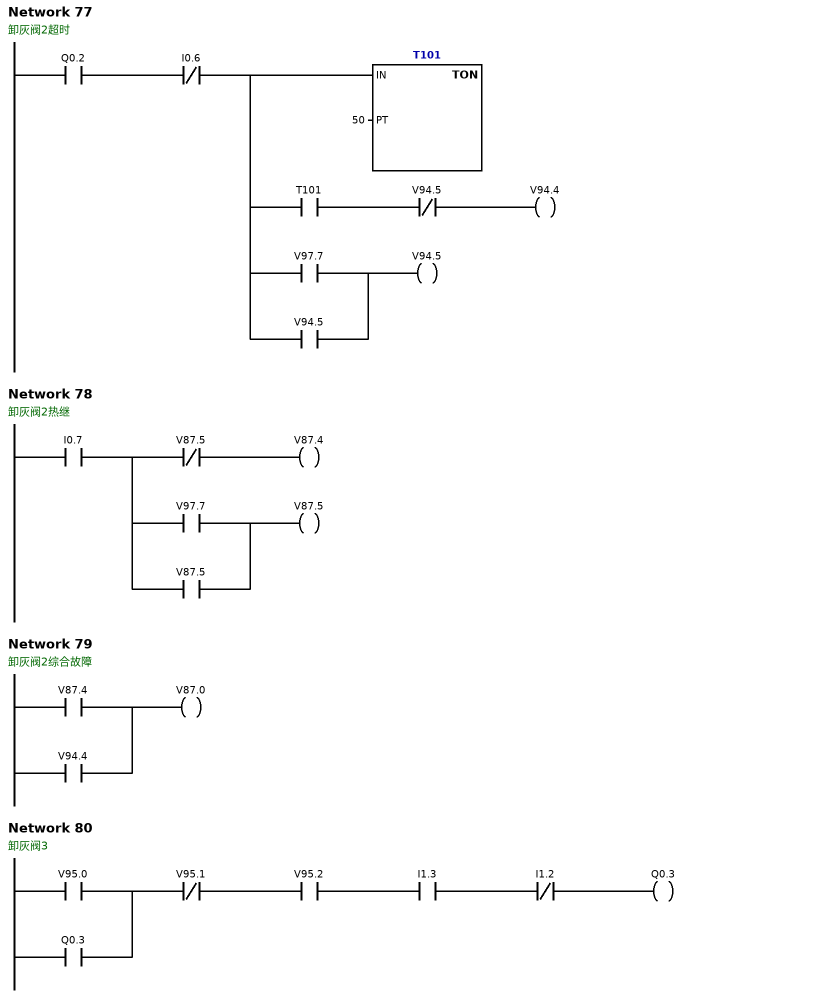
Network 77
// 卸灰阀2超时
LD     Q0.2
AN     I0.6
LPS
TON    T101, 50
A      T101
AN     V94.5
=      V94.4
LPP
LD     V97.7
O      V94.5
ALD
=      V94.5
Network 78
// 卸灰阀2热继
LD     I0.7
LPS
AN     V87.5
=      V87.4
LPP
LD     V97.7
O      V87.5
ALD
=      V87.5
Network 79
// 卸灰阀2综合故障
LD     V87.4
O      V94.4
=      V87.0
Network 80
// 卸灰阀3
LD     V95.0
O      Q0.3
AN     V95.1
A      V95.2
A      I1.3
AN     I1.2
=      Q0.3
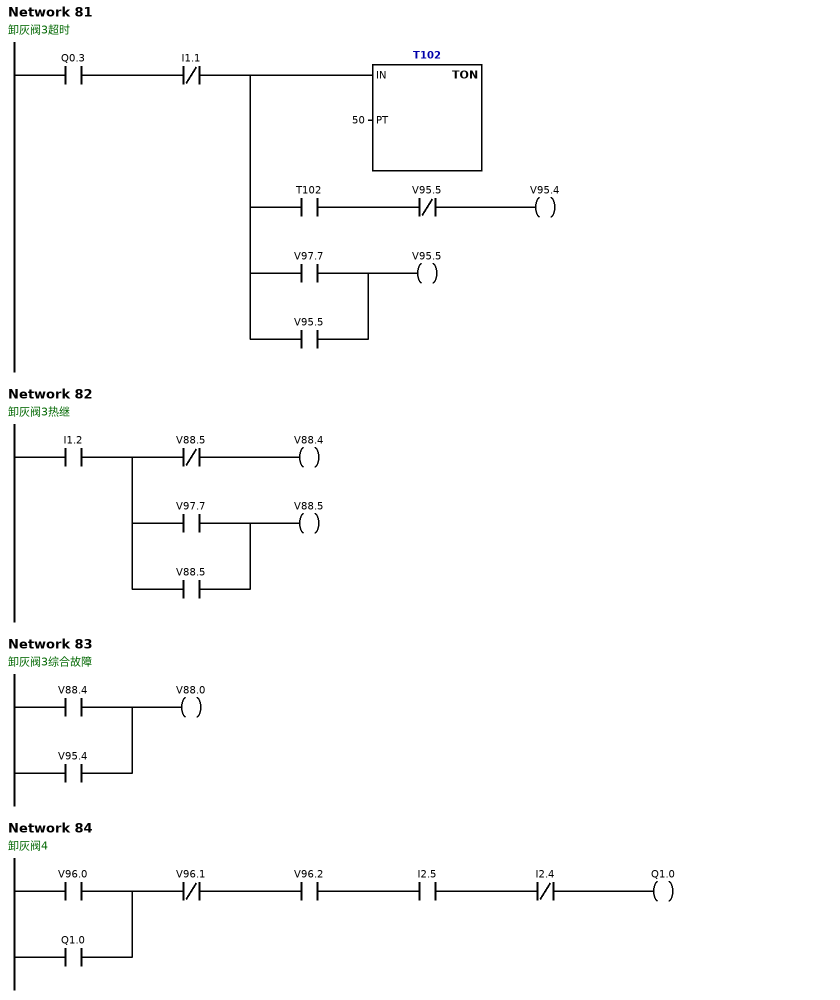
Network 81
// 卸灰阀3超时
LD     Q0.3
AN     I1.1
LPS
TON    T102, 50
A      T102
AN     V95.5
=      V95.4
LPP
LD     V97.7
O      V95.5
ALD
=      V95.5
Network 82
// 卸灰阀3热继
LD     I1.2
LPS
AN     V88.5
=      V88.4
LPP
LD     V97.7
O      V88.5
ALD
=      V88.5
Network 83
// 卸灰阀3综合故障
LD     V88.4
O      V95.4
=      V88.0
Network 84
// 卸灰阀4
LD     V96.0
O      Q1.0
AN     V96.1
A      V96.2
A      I2.5
AN     I2.4
=      Q1.0
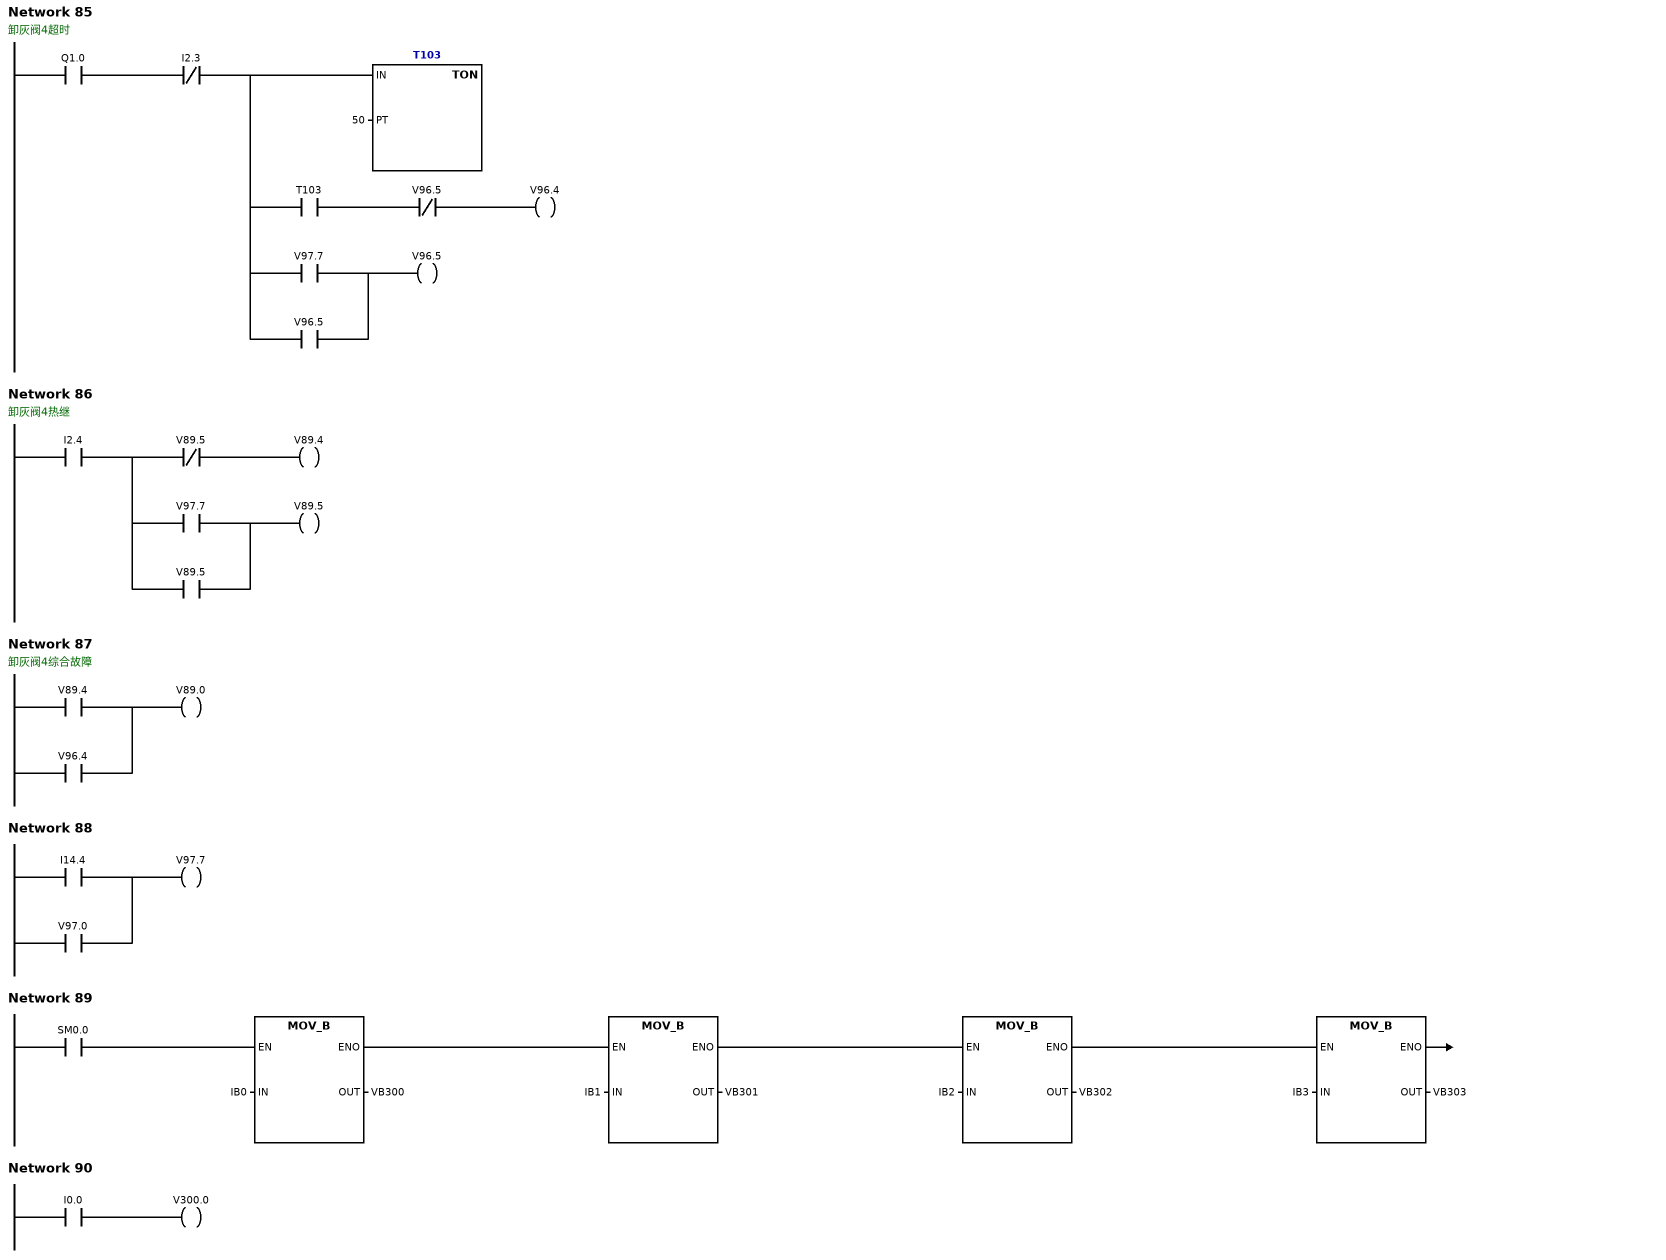
Network 85
// 卸灰阀4超时
LD     Q1.0
AN     I2.3
LPS
TON    T103, 50
A      T103
AN     V96.5
=      V96.4
LPP
LD     V97.7
O      V96.5
ALD
=      V96.5
Network 86
// 卸灰阀4热继
LD     I2.4
LPS
AN     V89.5
=      V89.4
LPP
LD     V97.7
O      V89.5
ALD
=      V89.5
Network 87
// 卸灰阀4综合故障
LD     V89.4
O      V96.4
=      V89.0
Network 88
LD     I14.4
O      V97.0
=      V97.7
Network 89
LD     SM0.0
MOVB   IB0, VB300
AENO
MOVB   IB1, VB301
AENO
MOVB   IB2, VB302
AENO
MOVB   IB3, VB303
Network 90
LD     I0.0
=      V300.0
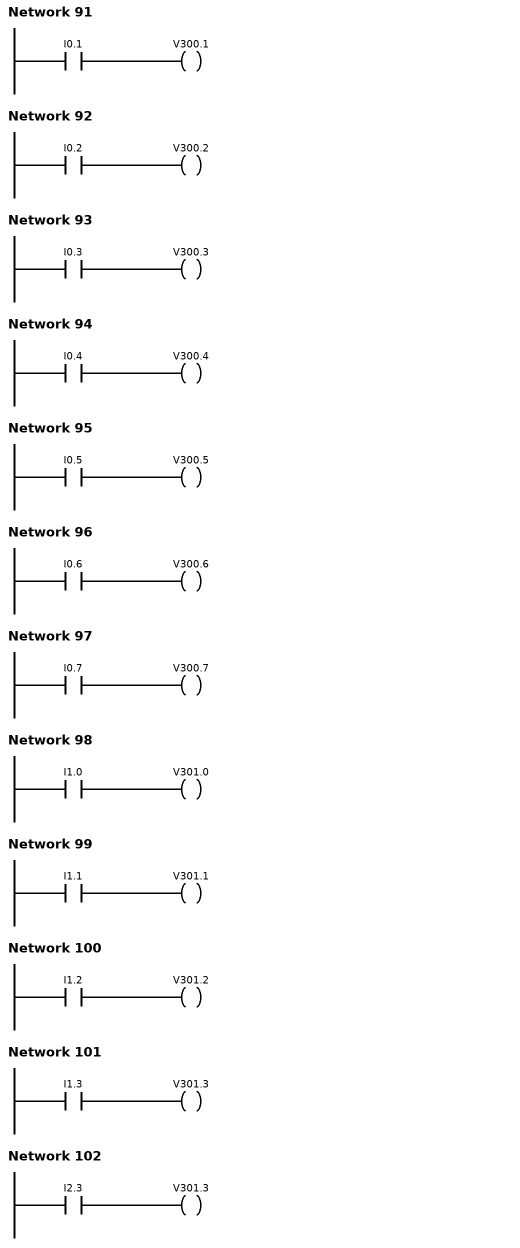
Network 91
// (network saved uncompiled; LAD cells follow)
// row 0: c0 -| |- I0.1  c1 -( ) V300.1
Network 92
// (network saved uncompiled; LAD cells follow)
// row 0: c0 -| |- I0.2  c1 -( ) V300.2
Network 93
// (network saved uncompiled; LAD cells follow)
// row 0: c0 -| |- I0.3  c1 -( ) V300.3
Network 94
// (network saved uncompiled; LAD cells follow)
// row 0: c0 -| |- I0.4  c1 -( ) V300.4
Network 95
// (network saved uncompiled; LAD cells follow)
// row 0: c0 -| |- I0.5  c1 -( ) V300.5
Network 96
// (network saved uncompiled; LAD cells follow)
// row 0: c0 -| |- I0.6  c1 -( ) V300.6
Network 97
// (network saved uncompiled; LAD cells follow)
// row 0: c0 -| |- I0.7  c1 -( ) V300.7
Network 98
// (network saved uncompiled; LAD cells follow)
// row 0: c0 -| |- I1.0  c1 -( ) V301.0
Network 99
// (network saved uncompiled; LAD cells follow)
// row 0: c0 -| |- I1.1  c1 -( ) V301.1
Network 100
// (network saved uncompiled; LAD cells follow)
// row 0: c0 -| |- I1.2  c1 -( ) V301.2
Network 101
// (network saved uncompiled; LAD cells follow)
// row 0: c0 -| |- I1.3  c1 -( ) V301.3
Network 102
// (network saved uncompiled; LAD cells follow)
// row 0: c0 -| |- I2.3  c1 -( ) V301.3
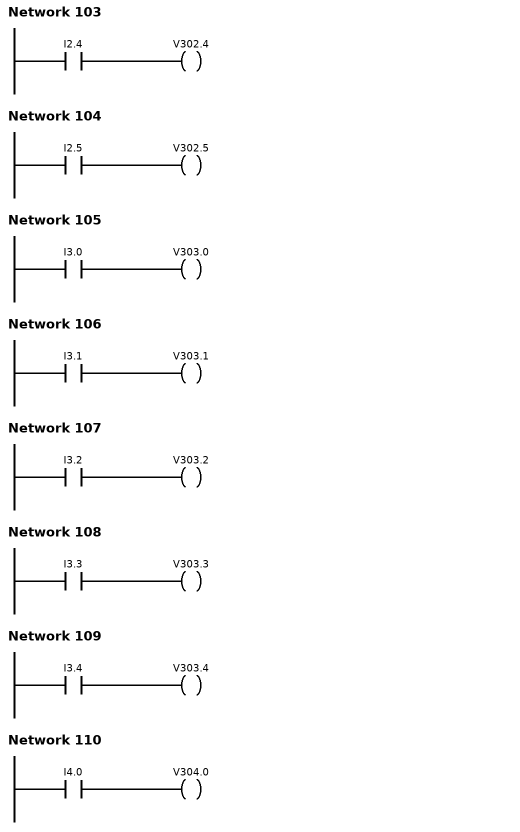
Network 103
// (network saved uncompiled; LAD cells follow)
// row 0: c0 -| |- I2.4  c1 -( ) V302.4
Network 104
// (network saved uncompiled; LAD cells follow)
// row 0: c0 -| |- I2.5  c1 -( ) V302.5
Network 105
// (network saved uncompiled; LAD cells follow)
// row 0: c0 -| |- I3.0  c1 -( ) V303.0
Network 106
// (network saved uncompiled; LAD cells follow)
// row 0: c0 -| |- I3.1  c1 -( ) V303.1
Network 107
// (network saved uncompiled; LAD cells follow)
// row 0: c0 -| |- I3.2  c1 -( ) V303.2
Network 108
// (network saved uncompiled; LAD cells follow)
// row 0: c0 -| |- I3.3  c1 -( ) V303.3
Network 109
// (network saved uncompiled; LAD cells follow)
// row 0: c0 -| |- I3.4  c1 -( ) V303.4
Network 110
// (network saved uncompiled; LAD cells follow)
// row 0: c0 -| |- I4.0  c1 -( ) V304.0
END_ORGANIZATION_BLOCK
